// TIA Portal V17 export
// export: Created 2025-05-08T13:17:33.0861985Z, ExportSetting WithDefaults, DisplayName Totally Integrated Automation Portal, DisplayVersion V17 Update 8, DisplayName TIA Portal Openness, DisplayVersion V17 Update 8, DisplayName TIA Portal Version Control Interface, DisplayVersion V17, DisplayName SINAMICS Startdrive Advanced, DisplayVersion V17 SP2, DisplayName SINAMICS Startdrive G110M, G120, G120C, G120D, G120P, G115D, DisplayVersion V17 SP2, DisplayName SINAMICS Startdrive G130, G150, S120, S150, SINAMICS MV, S210, DisplayVersion V17 SP2, DisplayName STEP 7 Professional, DisplayVersion V17 Update 8, DisplayName SINUMERIK ONE STEP 7 Toolbox, DisplayVersion V17 Update 12, DisplayName SINUMERIK 840D sl STEP 7 Toolbox, DisplayVersion V17 Update 12, DisplayName STEP 7 Safety, DisplayVersion V17 Update 6, DisplayName WinCC Advanced, DisplayVersion V17 Update 8
FUNCTION "FC3500_UNIT_2_FIXTURES" : Void   // FC3500, LAD
TITLE = FIXTURE 1
{ S7_Optimized_Access := 'FALSE' }
AUTHOR : ETXETAR
VERSION : 1.0
// stored: AutoNumber false, IsIECCheckEnabled false, SetENOAutomatically false, UDAEnableTagReadback false
   VAR CONSTANT
      FC_NUMBER : DInt := 2500;
   END_VAR
BEGIN

REGION Network 1: CALL FB2500 FIXTURE 1 UNIT 2 CLADDING
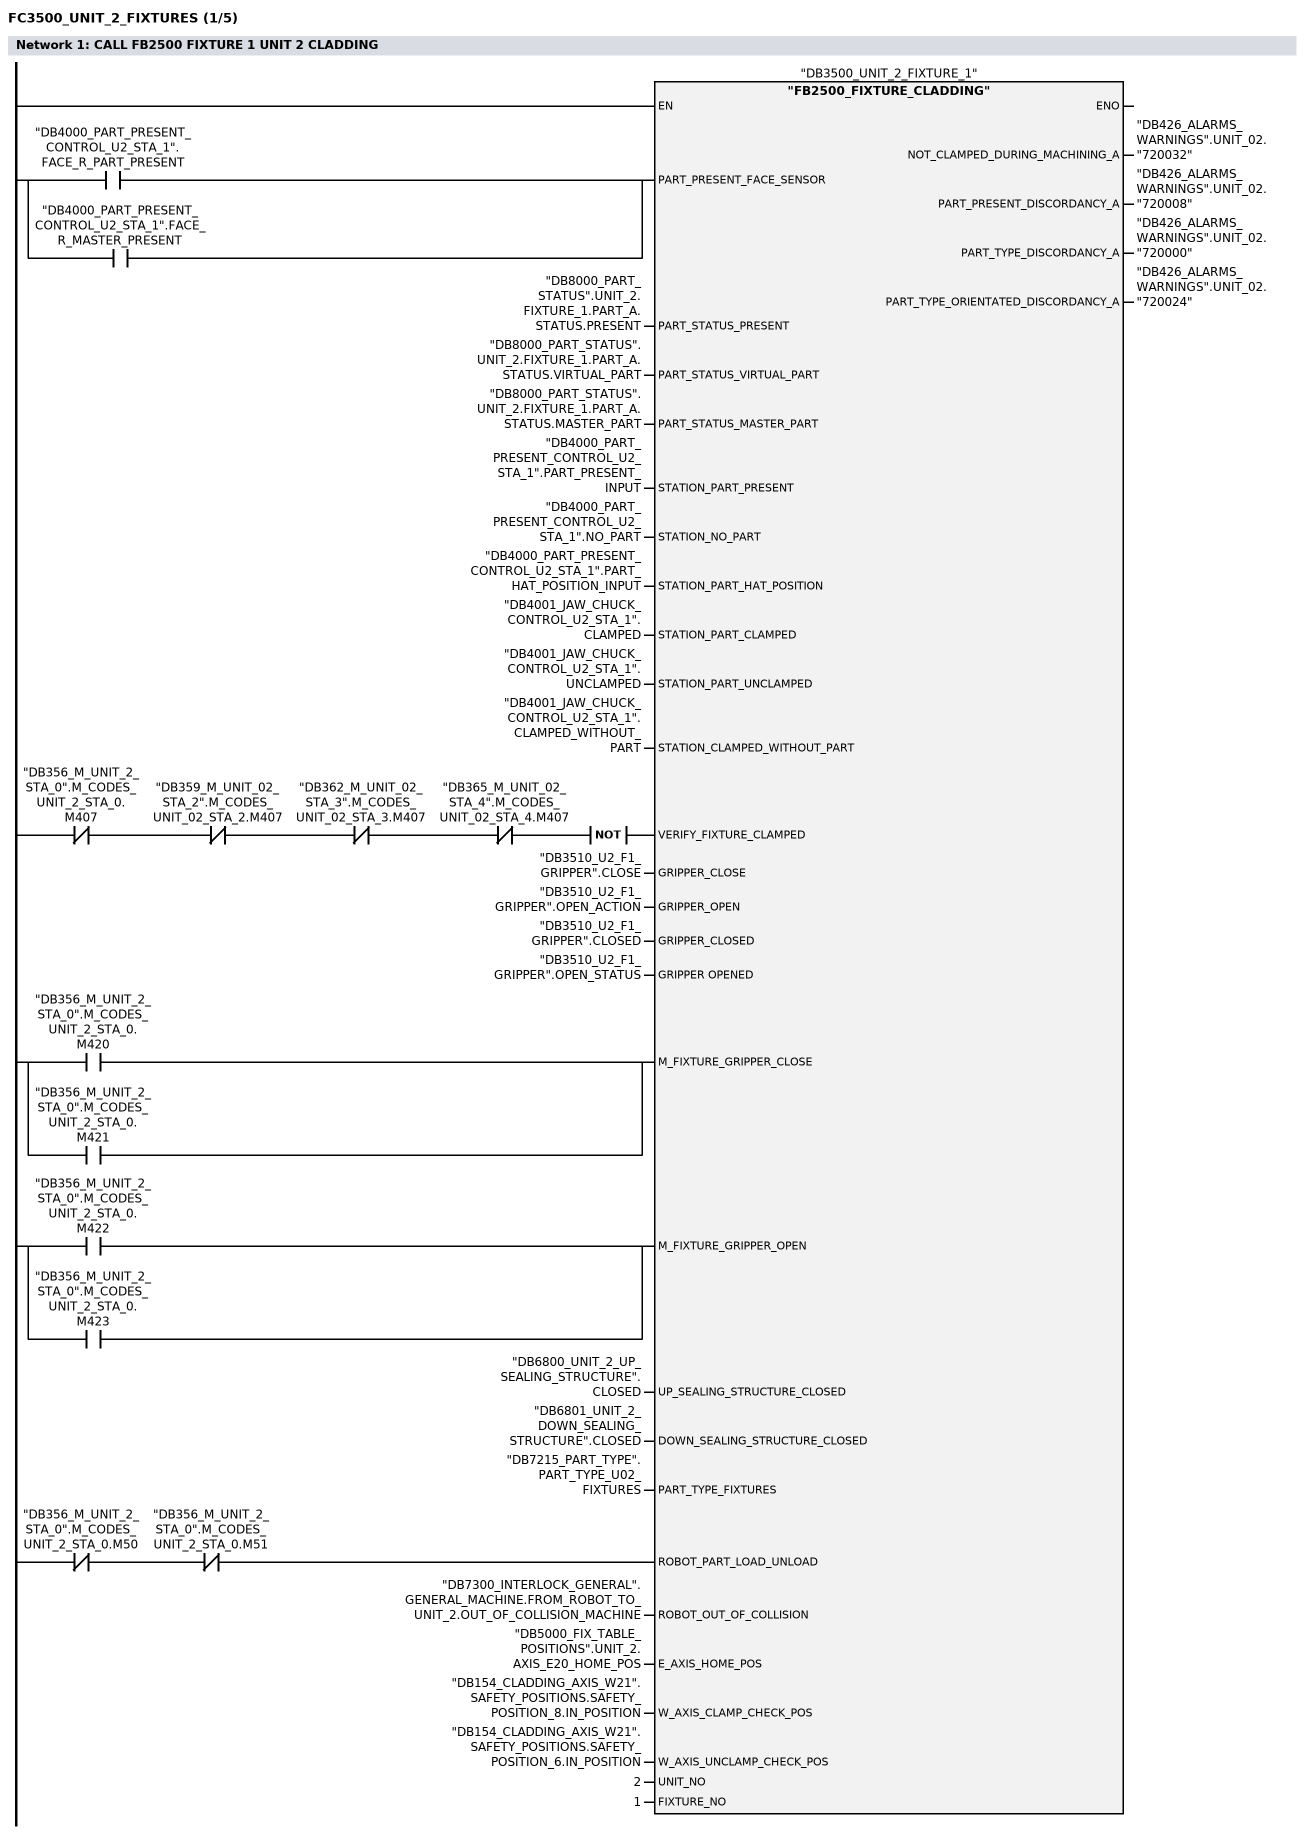
   RUNG wire#powerrail
      "DB3500_UNIT_2_FIXTURE_1"(PART_PRESENT_FACE_SENSOR := wire#w1, VERIFY_FIXTURE_CLAMPED := wire#w2, M_FIXTURE_GRIPPER_CLOSE := wire#w3, M_FIXTURE_GRIPPER_OPEN := wire#w4, ROBOT_PART_LOAD_UNLOAD := wire#w5, PART_STATUS_PRESENT := "DB8000_PART_STATUS".UNIT_2.FIXTURE_1.PART_A.STATUS.PRESENT, PART_STATUS_VIRTUAL_PART := "DB8000_PART_STATUS".UNIT_2.FIXTURE_1.PART_A.STATUS.VIRTUAL_PART, PART_STATUS_MASTER_PART := "DB8000_PART_STATUS".UNIT_2.FIXTURE_1.PART_A.STATUS.MASTER_PART, STATION_PART_PRESENT := "DB4000_PART_PRESENT_CONTROL_U2_STA_1".PART_PRESENT_INPUT, STATION_NO_PART := "DB4000_PART_PRESENT_CONTROL_U2_STA_1".NO_PART, STATION_PART_HAT_POSITION := "DB4000_PART_PRESENT_CONTROL_U2_STA_1".PART_HAT_POSITION_INPUT, STATION_PART_CLAMPED := "DB4001_JAW_CHUCK_CONTROL_U2_STA_1".CLAMPED, STATION_PART_UNCLAMPED := "DB4001_JAW_CHUCK_CONTROL_U2_STA_1".UNCLAMPED, STATION_CLAMPED_WITHOUT_PART := "DB4001_JAW_CHUCK_CONTROL_U2_STA_1".CLAMPED_WITHOUT_PART, GRIPPER_CLOSE := "DB3510_U2_F1_GRIPPER".CLOSE, GRIPPER_OPEN := "DB3510_U2_F1_GRIPPER".OPEN_ACTION, GRIPPER_CLOSED := "DB3510_U2_F1_GRIPPER".CLOSED, "GRIPPER OPENED" := "DB3510_U2_F1_GRIPPER".OPEN_STATUS, UP_SEALING_STRUCTURE_CLOSED := "DB6800_UNIT_2_UP_SEALING_STRUCTURE".CLOSED, DOWN_SEALING_STRUCTURE_CLOSED := "DB6801_UNIT_2_DOWN_SEALING_STRUCTURE".CLOSED, PART_TYPE_FIXTURES := "DB7215_PART_TYPE".PART_TYPE_U02_FIXTURES, ROBOT_OUT_OF_COLLISION := "DB7300_INTERLOCK_GENERAL".GENERAL_MACHINE.FROM_ROBOT_TO_UNIT_2.OUT_OF_COLLISION_MACHINE, E_AXIS_HOME_POS := "DB5000_FIX_TABLE_POSITIONS".UNIT_2.AXIS_E20_HOME_POS, W_AXIS_CLAMP_CHECK_POS := "DB154_CLADDING_AXIS_W21".SAFETY_POSITIONS.SAFETY_POSITION_8.IN_POSITION, W_AXIS_UNCLAMP_CHECK_POS := "DB154_CLADDING_AXIS_W21".SAFETY_POSITIONS.SAFETY_POSITION_6.IN_POSITION, UNIT_NO := 2, FIXTURE_NO := 1, NOT_CLAMPED_DURING_MACHINING_A => "DB426_ALARMS_WARNINGS".UNIT_02."720032", PART_PRESENT_DISCORDANCY_A => "DB426_ALARMS_WARNINGS".UNIT_02."720008", PART_TYPE_DISCORDANCY_A => "DB426_ALARMS_WARNINGS".UNIT_02."720000", PART_TYPE_ORIENTATED_DISCORDANCY_A => "DB426_ALARMS_WARNINGS".UNIT_02."720024")
   END_RUNG
   RUNG wire#powerrail
      Contact( "DB4000_PART_PRESENT_CONTROL_U2_STA_1".FACE_R_PART_PRESENT )
   END_RUNG wire#w1
   RUNG wire#powerrail
      Contact( "DB4000_PART_PRESENT_CONTROL_U2_STA_1".FACE_R_MASTER_PRESENT )
   END_RUNG wire#w1
   RUNG wire#powerrail
      I_Contact( "DB356_M_UNIT_2_STA_0".M_CODES_UNIT_2_STA_0.M407 )
      I_Contact( "DB359_M_UNIT_02_STA_2".M_CODES_UNIT_02_STA_2.M407 )
      I_Contact( "DB362_M_UNIT_02_STA_3".M_CODES_UNIT_02_STA_3.M407 )
      I_Contact( "DB365_M_UNIT_02_STA_4".M_CODES_UNIT_02_STA_4.M407 )
      Not()
   END_RUNG wire#w2
   RUNG wire#powerrail
      Contact( "DB356_M_UNIT_2_STA_0".M_CODES_UNIT_2_STA_0.M420 )
   END_RUNG wire#w3
   RUNG wire#powerrail
      Contact( "DB356_M_UNIT_2_STA_0".M_CODES_UNIT_2_STA_0.M421 )
   END_RUNG wire#w3
   RUNG wire#powerrail
      Contact( "DB356_M_UNIT_2_STA_0".M_CODES_UNIT_2_STA_0.M422 )
   END_RUNG wire#w4
   RUNG wire#powerrail
      Contact( "DB356_M_UNIT_2_STA_0".M_CODES_UNIT_2_STA_0.M423 )
   END_RUNG wire#w4
   RUNG wire#powerrail
      I_Contact( "DB356_M_UNIT_2_STA_0".M_CODES_UNIT_2_STA_0.M50 )
      I_Contact( "DB356_M_UNIT_2_STA_0".M_CODES_UNIT_2_STA_0.M51 )
   END_RUNG wire#w5
   // the same network as SCL:
   "DB3500_UNIT_2_FIXTURE_1"(PART_PRESENT_FACE_SENSOR := "DB4000_PART_PRESENT_CONTROL_U2_STA_1".FACE_R_PART_PRESENT OR "DB4000_PART_PRESENT_CONTROL_U2_STA_1".FACE_R_MASTER_PRESENT,   // "FB2500_FIXTURE_CLADDING"
                           PART_STATUS_PRESENT := "DB8000_PART_STATUS".UNIT_2.FIXTURE_1.PART_A.STATUS.PRESENT,
                           PART_STATUS_VIRTUAL_PART := "DB8000_PART_STATUS".UNIT_2.FIXTURE_1.PART_A.STATUS.VIRTUAL_PART,
                           PART_STATUS_MASTER_PART := "DB8000_PART_STATUS".UNIT_2.FIXTURE_1.PART_A.STATUS.MASTER_PART,
                           STATION_PART_PRESENT := "DB4000_PART_PRESENT_CONTROL_U2_STA_1".PART_PRESENT_INPUT,
                           STATION_NO_PART := "DB4000_PART_PRESENT_CONTROL_U2_STA_1".NO_PART,
                           STATION_PART_HAT_POSITION := "DB4000_PART_PRESENT_CONTROL_U2_STA_1".PART_HAT_POSITION_INPUT,
                           STATION_PART_CLAMPED := "DB4001_JAW_CHUCK_CONTROL_U2_STA_1".CLAMPED,
                           STATION_PART_UNCLAMPED := "DB4001_JAW_CHUCK_CONTROL_U2_STA_1".UNCLAMPED,
                           STATION_CLAMPED_WITHOUT_PART := "DB4001_JAW_CHUCK_CONTROL_U2_STA_1".CLAMPED_WITHOUT_PART,
                           VERIFY_FIXTURE_CLAMPED := NOT (NOT "DB356_M_UNIT_2_STA_0".M_CODES_UNIT_2_STA_0.M407 AND NOT "DB359_M_UNIT_02_STA_2".M_CODES_UNIT_02_STA_2.M407 AND NOT "DB362_M_UNIT_02_STA_3".M_CODES_UNIT_02_STA_3.M407 AND NOT "DB365_M_UNIT_02_STA_4".M_CODES_UNIT_02_STA_4.M407),
                           GRIPPER_CLOSE := "DB3510_U2_F1_GRIPPER".CLOSE,
                           GRIPPER_OPEN := "DB3510_U2_F1_GRIPPER".OPEN_ACTION,
                           GRIPPER_CLOSED := "DB3510_U2_F1_GRIPPER".CLOSED,
                           "GRIPPER OPENED" := "DB3510_U2_F1_GRIPPER".OPEN_STATUS,
                           M_FIXTURE_GRIPPER_CLOSE := "DB356_M_UNIT_2_STA_0".M_CODES_UNIT_2_STA_0.M420 OR "DB356_M_UNIT_2_STA_0".M_CODES_UNIT_2_STA_0.M421,
                           M_FIXTURE_GRIPPER_OPEN := "DB356_M_UNIT_2_STA_0".M_CODES_UNIT_2_STA_0.M422 OR "DB356_M_UNIT_2_STA_0".M_CODES_UNIT_2_STA_0.M423,
                           UP_SEALING_STRUCTURE_CLOSED := "DB6800_UNIT_2_UP_SEALING_STRUCTURE".CLOSED,
                           DOWN_SEALING_STRUCTURE_CLOSED := "DB6801_UNIT_2_DOWN_SEALING_STRUCTURE".CLOSED,
                           PART_TYPE_FIXTURES := "DB7215_PART_TYPE".PART_TYPE_U02_FIXTURES,
                           ROBOT_PART_LOAD_UNLOAD := NOT "DB356_M_UNIT_2_STA_0".M_CODES_UNIT_2_STA_0.M50 AND NOT "DB356_M_UNIT_2_STA_0".M_CODES_UNIT_2_STA_0.M51,
                           ROBOT_OUT_OF_COLLISION := "DB7300_INTERLOCK_GENERAL".GENERAL_MACHINE.FROM_ROBOT_TO_UNIT_2.OUT_OF_COLLISION_MACHINE,
                           E_AXIS_HOME_POS := "DB5000_FIX_TABLE_POSITIONS".UNIT_2.AXIS_E20_HOME_POS,
                           W_AXIS_CLAMP_CHECK_POS := "DB154_CLADDING_AXIS_W21".SAFETY_POSITIONS.SAFETY_POSITION_8.IN_POSITION,
                           W_AXIS_UNCLAMP_CHECK_POS := "DB154_CLADDING_AXIS_W21".SAFETY_POSITIONS.SAFETY_POSITION_6.IN_POSITION,
                           UNIT_NO := 2,
                           FIXTURE_NO := 1,
                           NOT_CLAMPED_DURING_MACHINING_A => "DB426_ALARMS_WARNINGS".UNIT_02."720032",
                           PART_PRESENT_DISCORDANCY_A => "DB426_ALARMS_WARNINGS".UNIT_02."720008",
                           PART_TYPE_DISCORDANCY_A => "DB426_ALARMS_WARNINGS".UNIT_02."720000",
                           PART_TYPE_ORIENTATED_DISCORDANCY_A => "DB426_ALARMS_WARNINGS".UNIT_02."720024");
END_REGION

REGION Network 2: CALL FB2600 FIXTURE 2 UNIT 2 CLADDING
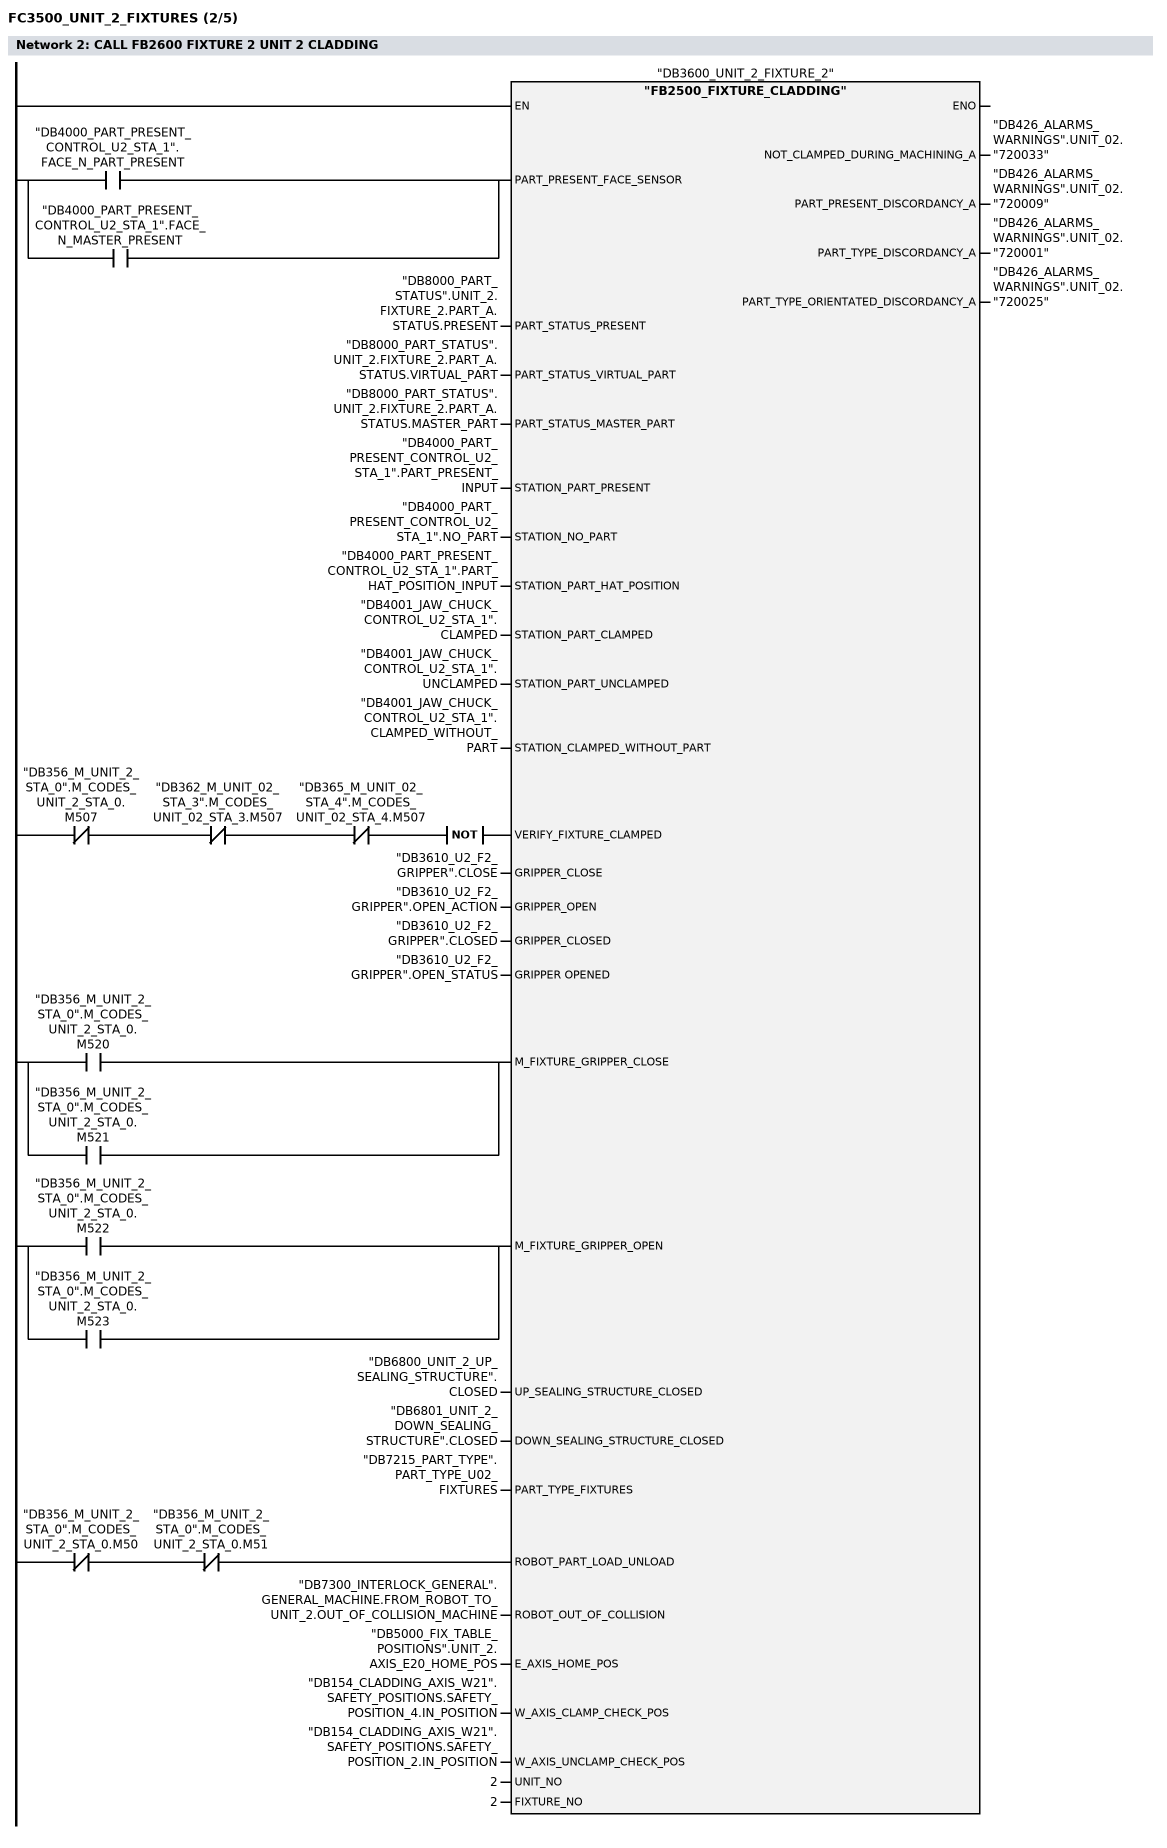
   RUNG wire#powerrail
      "DB3600_UNIT_2_FIXTURE_2"(PART_PRESENT_FACE_SENSOR := wire#w1, VERIFY_FIXTURE_CLAMPED := wire#w2, M_FIXTURE_GRIPPER_CLOSE := wire#w3, M_FIXTURE_GRIPPER_OPEN := wire#w4, ROBOT_PART_LOAD_UNLOAD := wire#w5, PART_STATUS_PRESENT := "DB8000_PART_STATUS".UNIT_2.FIXTURE_2.PART_A.STATUS.PRESENT, PART_STATUS_VIRTUAL_PART := "DB8000_PART_STATUS".UNIT_2.FIXTURE_2.PART_A.STATUS.VIRTUAL_PART, PART_STATUS_MASTER_PART := "DB8000_PART_STATUS".UNIT_2.FIXTURE_2.PART_A.STATUS.MASTER_PART, STATION_PART_PRESENT := "DB4000_PART_PRESENT_CONTROL_U2_STA_1".PART_PRESENT_INPUT, STATION_NO_PART := "DB4000_PART_PRESENT_CONTROL_U2_STA_1".NO_PART, STATION_PART_HAT_POSITION := "DB4000_PART_PRESENT_CONTROL_U2_STA_1".PART_HAT_POSITION_INPUT, STATION_PART_CLAMPED := "DB4001_JAW_CHUCK_CONTROL_U2_STA_1".CLAMPED, STATION_PART_UNCLAMPED := "DB4001_JAW_CHUCK_CONTROL_U2_STA_1".UNCLAMPED, STATION_CLAMPED_WITHOUT_PART := "DB4001_JAW_CHUCK_CONTROL_U2_STA_1".CLAMPED_WITHOUT_PART, GRIPPER_CLOSE := "DB3610_U2_F2_GRIPPER".CLOSE, GRIPPER_OPEN := "DB3610_U2_F2_GRIPPER".OPEN_ACTION, GRIPPER_CLOSED := "DB3610_U2_F2_GRIPPER".CLOSED, "GRIPPER OPENED" := "DB3610_U2_F2_GRIPPER".OPEN_STATUS, UP_SEALING_STRUCTURE_CLOSED := "DB6800_UNIT_2_UP_SEALING_STRUCTURE".CLOSED, DOWN_SEALING_STRUCTURE_CLOSED := "DB6801_UNIT_2_DOWN_SEALING_STRUCTURE".CLOSED, PART_TYPE_FIXTURES := "DB7215_PART_TYPE".PART_TYPE_U02_FIXTURES, ROBOT_OUT_OF_COLLISION := "DB7300_INTERLOCK_GENERAL".GENERAL_MACHINE.FROM_ROBOT_TO_UNIT_2.OUT_OF_COLLISION_MACHINE, E_AXIS_HOME_POS := "DB5000_FIX_TABLE_POSITIONS".UNIT_2.AXIS_E20_HOME_POS, W_AXIS_CLAMP_CHECK_POS := "DB154_CLADDING_AXIS_W21".SAFETY_POSITIONS.SAFETY_POSITION_4.IN_POSITION, W_AXIS_UNCLAMP_CHECK_POS := "DB154_CLADDING_AXIS_W21".SAFETY_POSITIONS.SAFETY_POSITION_2.IN_POSITION, UNIT_NO := 2, FIXTURE_NO := 2, NOT_CLAMPED_DURING_MACHINING_A => "DB426_ALARMS_WARNINGS".UNIT_02."720033", PART_PRESENT_DISCORDANCY_A => "DB426_ALARMS_WARNINGS".UNIT_02."720009", PART_TYPE_DISCORDANCY_A => "DB426_ALARMS_WARNINGS".UNIT_02."720001", PART_TYPE_ORIENTATED_DISCORDANCY_A => "DB426_ALARMS_WARNINGS".UNIT_02."720025")
   END_RUNG
   RUNG wire#powerrail
      Contact( "DB4000_PART_PRESENT_CONTROL_U2_STA_1".FACE_N_PART_PRESENT )
   END_RUNG wire#w1
   RUNG wire#powerrail
      Contact( "DB4000_PART_PRESENT_CONTROL_U2_STA_1".FACE_N_MASTER_PRESENT )
   END_RUNG wire#w1
   RUNG wire#powerrail
      I_Contact( "DB356_M_UNIT_2_STA_0".M_CODES_UNIT_2_STA_0.M507 )
      I_Contact( "DB362_M_UNIT_02_STA_3".M_CODES_UNIT_02_STA_3.M507 )
      I_Contact( "DB365_M_UNIT_02_STA_4".M_CODES_UNIT_02_STA_4.M507 )
      Not()
   END_RUNG wire#w2
   RUNG wire#powerrail
      Contact( "DB356_M_UNIT_2_STA_0".M_CODES_UNIT_2_STA_0.M520 )
   END_RUNG wire#w3
   RUNG wire#powerrail
      Contact( "DB356_M_UNIT_2_STA_0".M_CODES_UNIT_2_STA_0.M521 )
   END_RUNG wire#w3
   RUNG wire#powerrail
      Contact( "DB356_M_UNIT_2_STA_0".M_CODES_UNIT_2_STA_0.M522 )
   END_RUNG wire#w4
   RUNG wire#powerrail
      Contact( "DB356_M_UNIT_2_STA_0".M_CODES_UNIT_2_STA_0.M523 )
   END_RUNG wire#w4
   RUNG wire#powerrail
      I_Contact( "DB356_M_UNIT_2_STA_0".M_CODES_UNIT_2_STA_0.M50 )
      I_Contact( "DB356_M_UNIT_2_STA_0".M_CODES_UNIT_2_STA_0.M51 )
   END_RUNG wire#w5
   // the same network as SCL:
   "DB3600_UNIT_2_FIXTURE_2"(PART_PRESENT_FACE_SENSOR := "DB4000_PART_PRESENT_CONTROL_U2_STA_1".FACE_N_PART_PRESENT OR "DB4000_PART_PRESENT_CONTROL_U2_STA_1".FACE_N_MASTER_PRESENT,   // "FB2500_FIXTURE_CLADDING"
                           PART_STATUS_PRESENT := "DB8000_PART_STATUS".UNIT_2.FIXTURE_2.PART_A.STATUS.PRESENT,
                           PART_STATUS_VIRTUAL_PART := "DB8000_PART_STATUS".UNIT_2.FIXTURE_2.PART_A.STATUS.VIRTUAL_PART,
                           PART_STATUS_MASTER_PART := "DB8000_PART_STATUS".UNIT_2.FIXTURE_2.PART_A.STATUS.MASTER_PART,
                           STATION_PART_PRESENT := "DB4000_PART_PRESENT_CONTROL_U2_STA_1".PART_PRESENT_INPUT,
                           STATION_NO_PART := "DB4000_PART_PRESENT_CONTROL_U2_STA_1".NO_PART,
                           STATION_PART_HAT_POSITION := "DB4000_PART_PRESENT_CONTROL_U2_STA_1".PART_HAT_POSITION_INPUT,
                           STATION_PART_CLAMPED := "DB4001_JAW_CHUCK_CONTROL_U2_STA_1".CLAMPED,
                           STATION_PART_UNCLAMPED := "DB4001_JAW_CHUCK_CONTROL_U2_STA_1".UNCLAMPED,
                           STATION_CLAMPED_WITHOUT_PART := "DB4001_JAW_CHUCK_CONTROL_U2_STA_1".CLAMPED_WITHOUT_PART,
                           VERIFY_FIXTURE_CLAMPED := NOT (NOT "DB356_M_UNIT_2_STA_0".M_CODES_UNIT_2_STA_0.M507 AND NOT "DB362_M_UNIT_02_STA_3".M_CODES_UNIT_02_STA_3.M507 AND NOT "DB365_M_UNIT_02_STA_4".M_CODES_UNIT_02_STA_4.M507),
                           GRIPPER_CLOSE := "DB3610_U2_F2_GRIPPER".CLOSE,
                           GRIPPER_OPEN := "DB3610_U2_F2_GRIPPER".OPEN_ACTION,
                           GRIPPER_CLOSED := "DB3610_U2_F2_GRIPPER".CLOSED,
                           "GRIPPER OPENED" := "DB3610_U2_F2_GRIPPER".OPEN_STATUS,
                           M_FIXTURE_GRIPPER_CLOSE := "DB356_M_UNIT_2_STA_0".M_CODES_UNIT_2_STA_0.M520 OR "DB356_M_UNIT_2_STA_0".M_CODES_UNIT_2_STA_0.M521,
                           M_FIXTURE_GRIPPER_OPEN := "DB356_M_UNIT_2_STA_0".M_CODES_UNIT_2_STA_0.M522 OR "DB356_M_UNIT_2_STA_0".M_CODES_UNIT_2_STA_0.M523,
                           UP_SEALING_STRUCTURE_CLOSED := "DB6800_UNIT_2_UP_SEALING_STRUCTURE".CLOSED,
                           DOWN_SEALING_STRUCTURE_CLOSED := "DB6801_UNIT_2_DOWN_SEALING_STRUCTURE".CLOSED,
                           PART_TYPE_FIXTURES := "DB7215_PART_TYPE".PART_TYPE_U02_FIXTURES,
                           ROBOT_PART_LOAD_UNLOAD := NOT "DB356_M_UNIT_2_STA_0".M_CODES_UNIT_2_STA_0.M50 AND NOT "DB356_M_UNIT_2_STA_0".M_CODES_UNIT_2_STA_0.M51,
                           ROBOT_OUT_OF_COLLISION := "DB7300_INTERLOCK_GENERAL".GENERAL_MACHINE.FROM_ROBOT_TO_UNIT_2.OUT_OF_COLLISION_MACHINE,
                           E_AXIS_HOME_POS := "DB5000_FIX_TABLE_POSITIONS".UNIT_2.AXIS_E20_HOME_POS,
                           W_AXIS_CLAMP_CHECK_POS := "DB154_CLADDING_AXIS_W21".SAFETY_POSITIONS.SAFETY_POSITION_4.IN_POSITION,
                           W_AXIS_UNCLAMP_CHECK_POS := "DB154_CLADDING_AXIS_W21".SAFETY_POSITIONS.SAFETY_POSITION_2.IN_POSITION,
                           UNIT_NO := 2,
                           FIXTURE_NO := 2,
                           NOT_CLAMPED_DURING_MACHINING_A => "DB426_ALARMS_WARNINGS".UNIT_02."720033",
                           PART_PRESENT_DISCORDANCY_A => "DB426_ALARMS_WARNINGS".UNIT_02."720009",
                           PART_TYPE_DISCORDANCY_A => "DB426_ALARMS_WARNINGS".UNIT_02."720001",
                           PART_TYPE_ORIENTATED_DISCORDANCY_A => "DB426_ALARMS_WARNINGS".UNIT_02."720025");
END_REGION

REGION Network 3: CALL FB2600 FIXTURE 3 UNIT 2 CLADDING
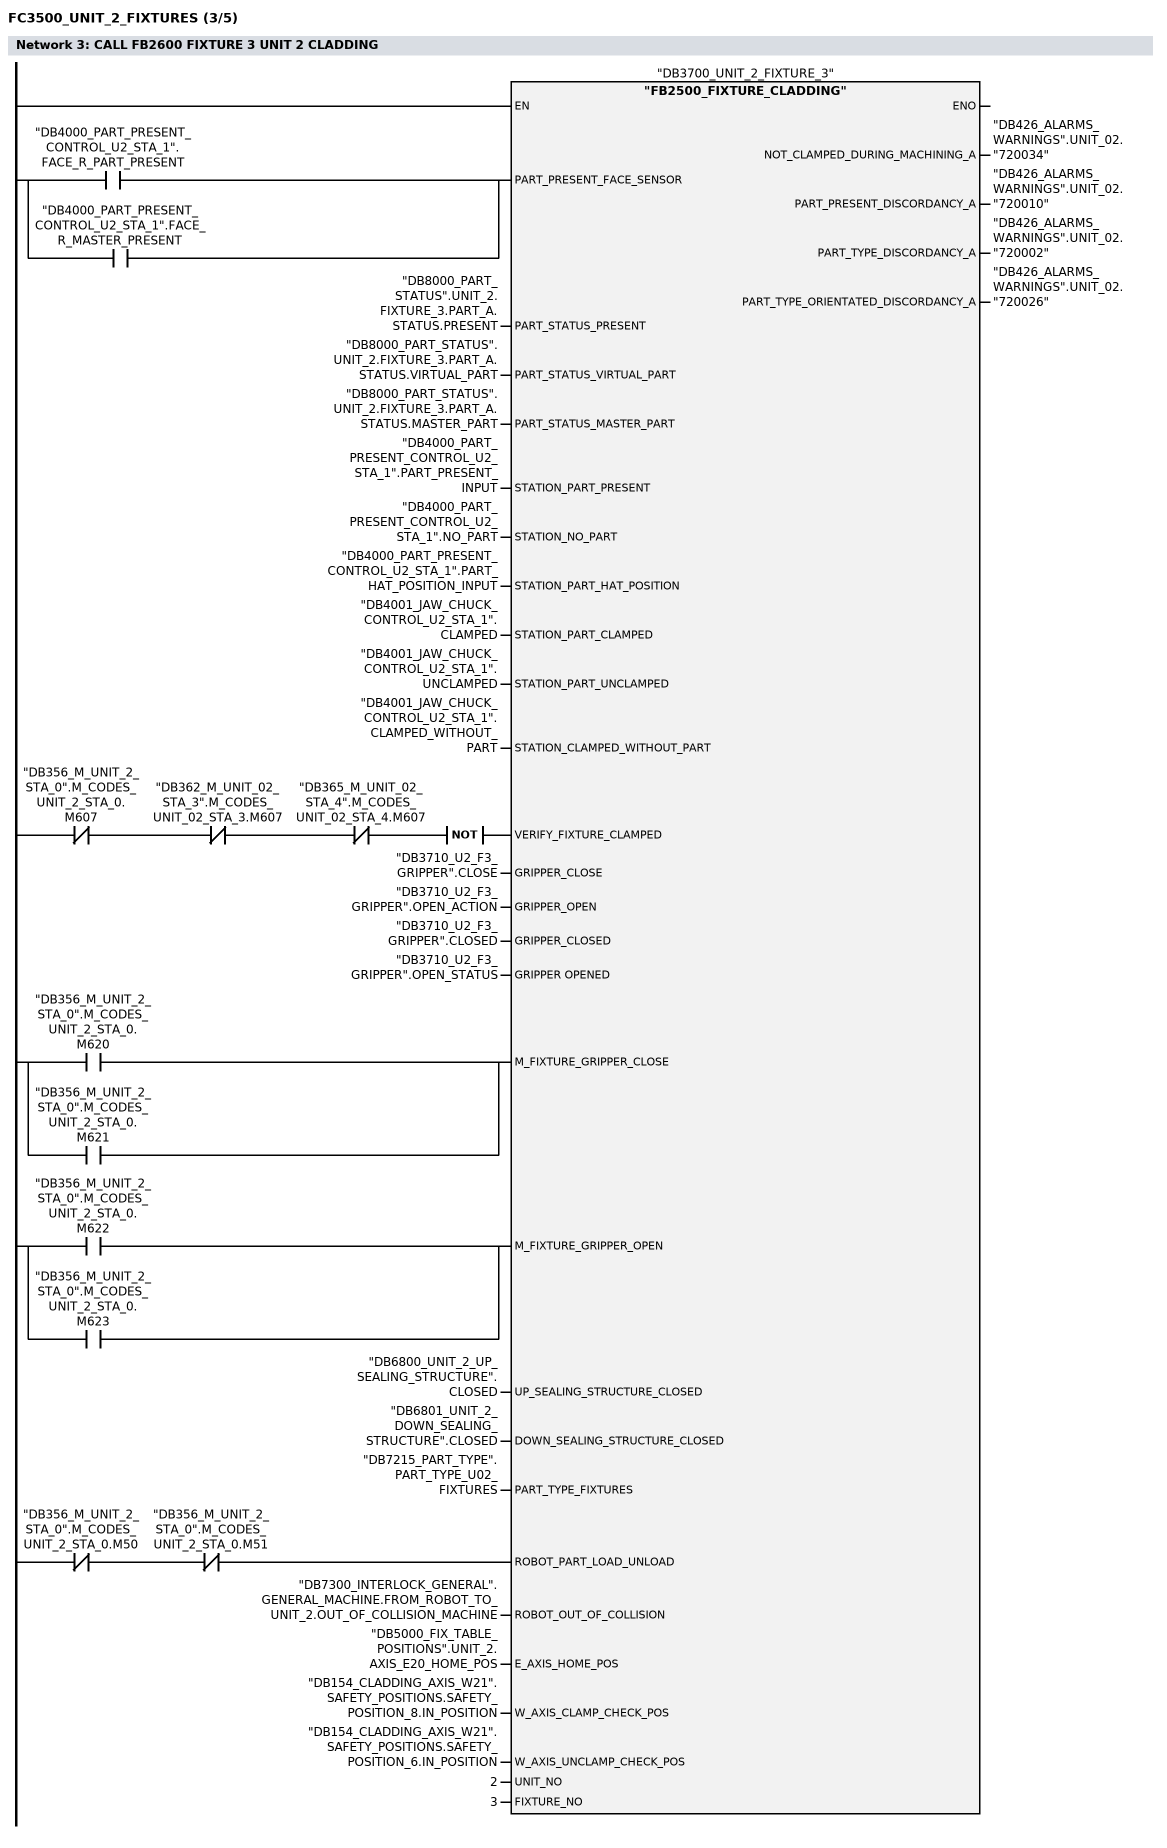
   RUNG wire#powerrail
      "DB3700_UNIT_2_FIXTURE_3"(PART_PRESENT_FACE_SENSOR := wire#w1, VERIFY_FIXTURE_CLAMPED := wire#w2, M_FIXTURE_GRIPPER_CLOSE := wire#w3, M_FIXTURE_GRIPPER_OPEN := wire#w4, ROBOT_PART_LOAD_UNLOAD := wire#w5, PART_STATUS_PRESENT := "DB8000_PART_STATUS".UNIT_2.FIXTURE_3.PART_A.STATUS.PRESENT, PART_STATUS_VIRTUAL_PART := "DB8000_PART_STATUS".UNIT_2.FIXTURE_3.PART_A.STATUS.VIRTUAL_PART, PART_STATUS_MASTER_PART := "DB8000_PART_STATUS".UNIT_2.FIXTURE_3.PART_A.STATUS.MASTER_PART, STATION_PART_PRESENT := "DB4000_PART_PRESENT_CONTROL_U2_STA_1".PART_PRESENT_INPUT, STATION_NO_PART := "DB4000_PART_PRESENT_CONTROL_U2_STA_1".NO_PART, STATION_PART_HAT_POSITION := "DB4000_PART_PRESENT_CONTROL_U2_STA_1".PART_HAT_POSITION_INPUT, STATION_PART_CLAMPED := "DB4001_JAW_CHUCK_CONTROL_U2_STA_1".CLAMPED, STATION_PART_UNCLAMPED := "DB4001_JAW_CHUCK_CONTROL_U2_STA_1".UNCLAMPED, STATION_CLAMPED_WITHOUT_PART := "DB4001_JAW_CHUCK_CONTROL_U2_STA_1".CLAMPED_WITHOUT_PART, GRIPPER_CLOSE := "DB3710_U2_F3_GRIPPER".CLOSE, GRIPPER_OPEN := "DB3710_U2_F3_GRIPPER".OPEN_ACTION, GRIPPER_CLOSED := "DB3710_U2_F3_GRIPPER".CLOSED, "GRIPPER OPENED" := "DB3710_U2_F3_GRIPPER".OPEN_STATUS, UP_SEALING_STRUCTURE_CLOSED := "DB6800_UNIT_2_UP_SEALING_STRUCTURE".CLOSED, DOWN_SEALING_STRUCTURE_CLOSED := "DB6801_UNIT_2_DOWN_SEALING_STRUCTURE".CLOSED, PART_TYPE_FIXTURES := "DB7215_PART_TYPE".PART_TYPE_U02_FIXTURES, ROBOT_OUT_OF_COLLISION := "DB7300_INTERLOCK_GENERAL".GENERAL_MACHINE.FROM_ROBOT_TO_UNIT_2.OUT_OF_COLLISION_MACHINE, E_AXIS_HOME_POS := "DB5000_FIX_TABLE_POSITIONS".UNIT_2.AXIS_E20_HOME_POS, W_AXIS_CLAMP_CHECK_POS := "DB154_CLADDING_AXIS_W21".SAFETY_POSITIONS.SAFETY_POSITION_8.IN_POSITION, W_AXIS_UNCLAMP_CHECK_POS := "DB154_CLADDING_AXIS_W21".SAFETY_POSITIONS.SAFETY_POSITION_6.IN_POSITION, UNIT_NO := 2, FIXTURE_NO := 3, NOT_CLAMPED_DURING_MACHINING_A => "DB426_ALARMS_WARNINGS".UNIT_02."720034", PART_PRESENT_DISCORDANCY_A => "DB426_ALARMS_WARNINGS".UNIT_02."720010", PART_TYPE_DISCORDANCY_A => "DB426_ALARMS_WARNINGS".UNIT_02."720002", PART_TYPE_ORIENTATED_DISCORDANCY_A => "DB426_ALARMS_WARNINGS".UNIT_02."720026")
   END_RUNG
   RUNG wire#powerrail
      Contact( "DB4000_PART_PRESENT_CONTROL_U2_STA_1".FACE_R_PART_PRESENT )
   END_RUNG wire#w1
   RUNG wire#powerrail
      Contact( "DB4000_PART_PRESENT_CONTROL_U2_STA_1".FACE_R_MASTER_PRESENT )
   END_RUNG wire#w1
   RUNG wire#powerrail
      I_Contact( "DB356_M_UNIT_2_STA_0".M_CODES_UNIT_2_STA_0.M607 )
      I_Contact( "DB362_M_UNIT_02_STA_3".M_CODES_UNIT_02_STA_3.M607 )
      I_Contact( "DB365_M_UNIT_02_STA_4".M_CODES_UNIT_02_STA_4.M607 )
      Not()
   END_RUNG wire#w2
   RUNG wire#powerrail
      Contact( "DB356_M_UNIT_2_STA_0".M_CODES_UNIT_2_STA_0.M620 )
   END_RUNG wire#w3
   RUNG wire#powerrail
      Contact( "DB356_M_UNIT_2_STA_0".M_CODES_UNIT_2_STA_0.M621 )
   END_RUNG wire#w3
   RUNG wire#powerrail
      Contact( "DB356_M_UNIT_2_STA_0".M_CODES_UNIT_2_STA_0.M622 )
   END_RUNG wire#w4
   RUNG wire#powerrail
      Contact( "DB356_M_UNIT_2_STA_0".M_CODES_UNIT_2_STA_0.M623 )
   END_RUNG wire#w4
   RUNG wire#powerrail
      I_Contact( "DB356_M_UNIT_2_STA_0".M_CODES_UNIT_2_STA_0.M50 )
      I_Contact( "DB356_M_UNIT_2_STA_0".M_CODES_UNIT_2_STA_0.M51 )
   END_RUNG wire#w5
   // the same network as SCL:
   "DB3700_UNIT_2_FIXTURE_3"(PART_PRESENT_FACE_SENSOR := "DB4000_PART_PRESENT_CONTROL_U2_STA_1".FACE_R_PART_PRESENT OR "DB4000_PART_PRESENT_CONTROL_U2_STA_1".FACE_R_MASTER_PRESENT,   // "FB2500_FIXTURE_CLADDING"
                           PART_STATUS_PRESENT := "DB8000_PART_STATUS".UNIT_2.FIXTURE_3.PART_A.STATUS.PRESENT,
                           PART_STATUS_VIRTUAL_PART := "DB8000_PART_STATUS".UNIT_2.FIXTURE_3.PART_A.STATUS.VIRTUAL_PART,
                           PART_STATUS_MASTER_PART := "DB8000_PART_STATUS".UNIT_2.FIXTURE_3.PART_A.STATUS.MASTER_PART,
                           STATION_PART_PRESENT := "DB4000_PART_PRESENT_CONTROL_U2_STA_1".PART_PRESENT_INPUT,
                           STATION_NO_PART := "DB4000_PART_PRESENT_CONTROL_U2_STA_1".NO_PART,
                           STATION_PART_HAT_POSITION := "DB4000_PART_PRESENT_CONTROL_U2_STA_1".PART_HAT_POSITION_INPUT,
                           STATION_PART_CLAMPED := "DB4001_JAW_CHUCK_CONTROL_U2_STA_1".CLAMPED,
                           STATION_PART_UNCLAMPED := "DB4001_JAW_CHUCK_CONTROL_U2_STA_1".UNCLAMPED,
                           STATION_CLAMPED_WITHOUT_PART := "DB4001_JAW_CHUCK_CONTROL_U2_STA_1".CLAMPED_WITHOUT_PART,
                           VERIFY_FIXTURE_CLAMPED := NOT (NOT "DB356_M_UNIT_2_STA_0".M_CODES_UNIT_2_STA_0.M607 AND NOT "DB362_M_UNIT_02_STA_3".M_CODES_UNIT_02_STA_3.M607 AND NOT "DB365_M_UNIT_02_STA_4".M_CODES_UNIT_02_STA_4.M607),
                           GRIPPER_CLOSE := "DB3710_U2_F3_GRIPPER".CLOSE,
                           GRIPPER_OPEN := "DB3710_U2_F3_GRIPPER".OPEN_ACTION,
                           GRIPPER_CLOSED := "DB3710_U2_F3_GRIPPER".CLOSED,
                           "GRIPPER OPENED" := "DB3710_U2_F3_GRIPPER".OPEN_STATUS,
                           M_FIXTURE_GRIPPER_CLOSE := "DB356_M_UNIT_2_STA_0".M_CODES_UNIT_2_STA_0.M620 OR "DB356_M_UNIT_2_STA_0".M_CODES_UNIT_2_STA_0.M621,
                           M_FIXTURE_GRIPPER_OPEN := "DB356_M_UNIT_2_STA_0".M_CODES_UNIT_2_STA_0.M622 OR "DB356_M_UNIT_2_STA_0".M_CODES_UNIT_2_STA_0.M623,
                           UP_SEALING_STRUCTURE_CLOSED := "DB6800_UNIT_2_UP_SEALING_STRUCTURE".CLOSED,
                           DOWN_SEALING_STRUCTURE_CLOSED := "DB6801_UNIT_2_DOWN_SEALING_STRUCTURE".CLOSED,
                           PART_TYPE_FIXTURES := "DB7215_PART_TYPE".PART_TYPE_U02_FIXTURES,
                           ROBOT_PART_LOAD_UNLOAD := NOT "DB356_M_UNIT_2_STA_0".M_CODES_UNIT_2_STA_0.M50 AND NOT "DB356_M_UNIT_2_STA_0".M_CODES_UNIT_2_STA_0.M51,
                           ROBOT_OUT_OF_COLLISION := "DB7300_INTERLOCK_GENERAL".GENERAL_MACHINE.FROM_ROBOT_TO_UNIT_2.OUT_OF_COLLISION_MACHINE,
                           E_AXIS_HOME_POS := "DB5000_FIX_TABLE_POSITIONS".UNIT_2.AXIS_E20_HOME_POS,
                           W_AXIS_CLAMP_CHECK_POS := "DB154_CLADDING_AXIS_W21".SAFETY_POSITIONS.SAFETY_POSITION_8.IN_POSITION,
                           W_AXIS_UNCLAMP_CHECK_POS := "DB154_CLADDING_AXIS_W21".SAFETY_POSITIONS.SAFETY_POSITION_6.IN_POSITION,
                           UNIT_NO := 2,
                           FIXTURE_NO := 3,
                           NOT_CLAMPED_DURING_MACHINING_A => "DB426_ALARMS_WARNINGS".UNIT_02."720034",
                           PART_PRESENT_DISCORDANCY_A => "DB426_ALARMS_WARNINGS".UNIT_02."720010",
                           PART_TYPE_DISCORDANCY_A => "DB426_ALARMS_WARNINGS".UNIT_02."720002",
                           PART_TYPE_ORIENTATED_DISCORDANCY_A => "DB426_ALARMS_WARNINGS".UNIT_02."720026");
END_REGION

REGION Network 4: CALL FB2600 FIXTURE 4 UNIT 2 CLADDING
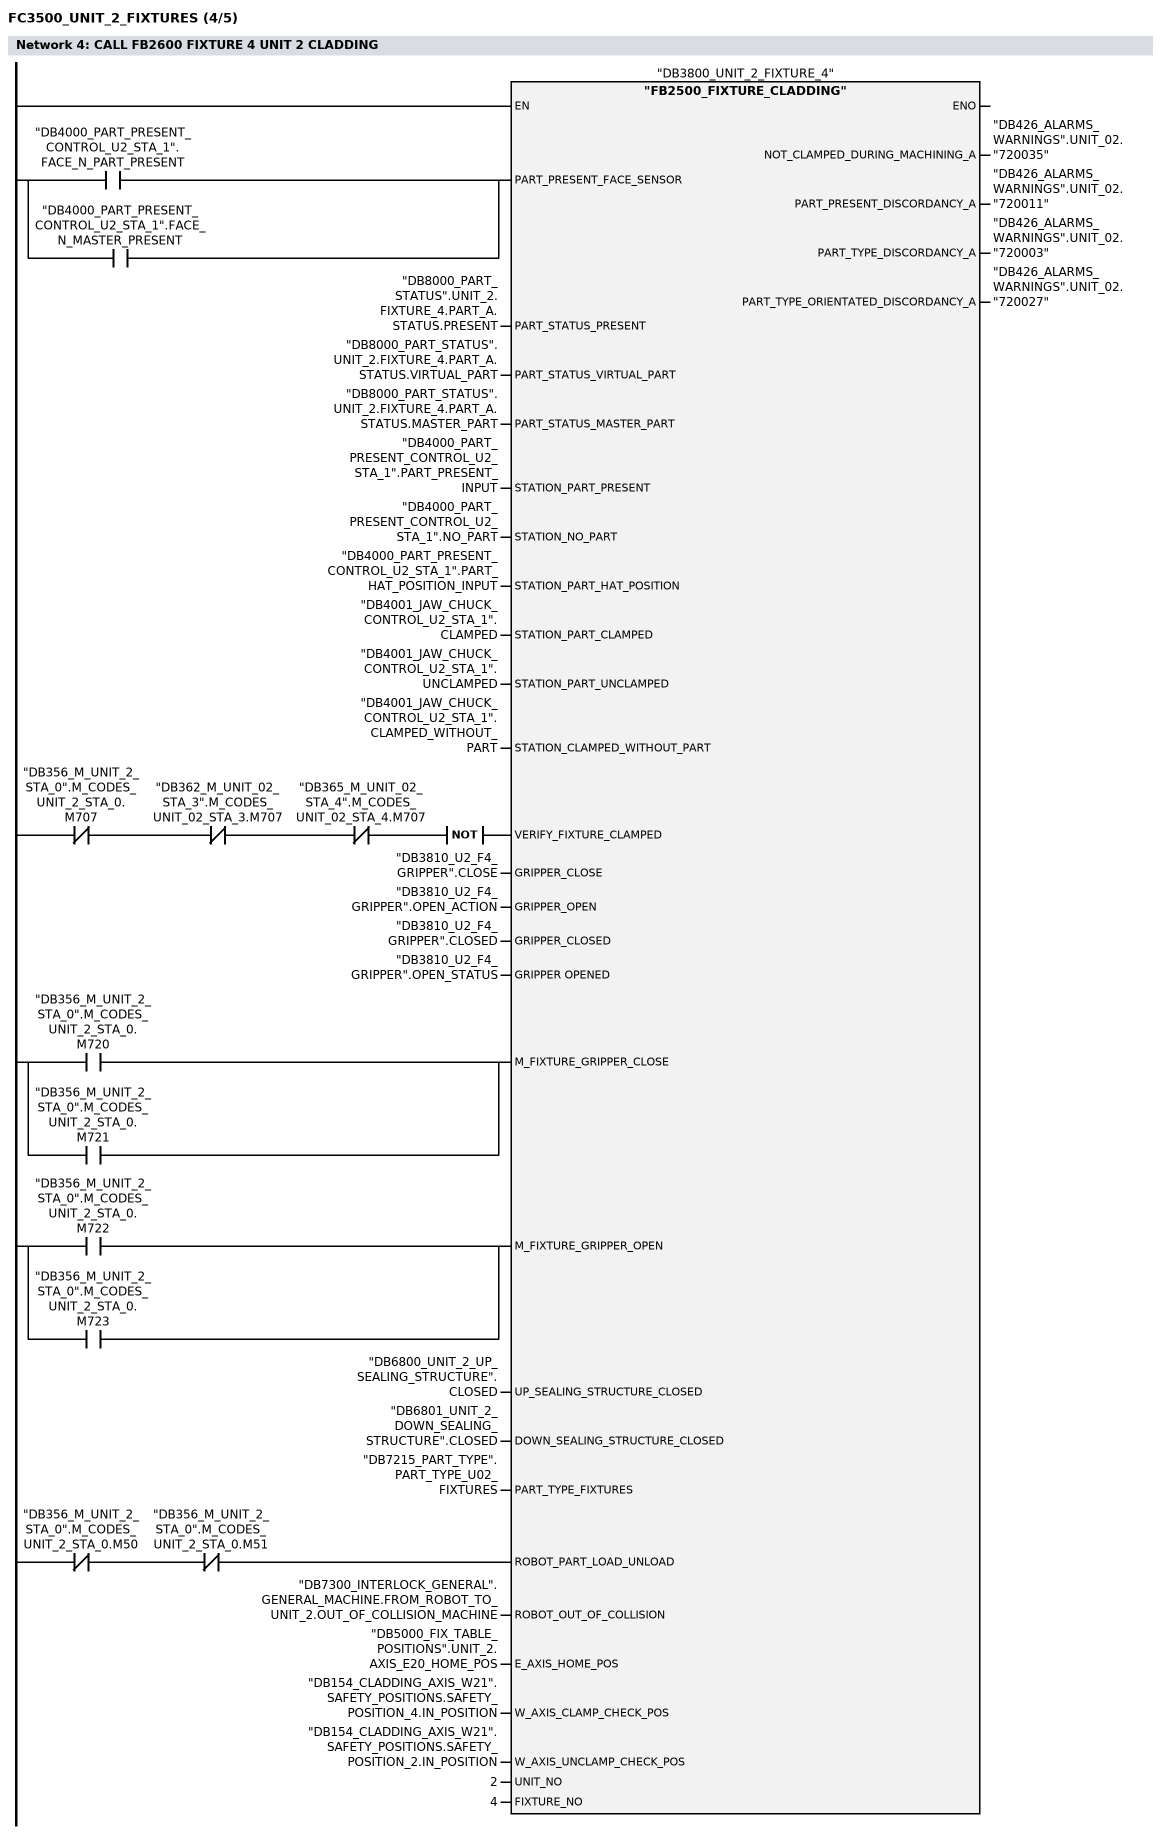
   RUNG wire#powerrail
      "DB3800_UNIT_2_FIXTURE_4"(PART_PRESENT_FACE_SENSOR := wire#w1, VERIFY_FIXTURE_CLAMPED := wire#w2, M_FIXTURE_GRIPPER_CLOSE := wire#w3, M_FIXTURE_GRIPPER_OPEN := wire#w4, ROBOT_PART_LOAD_UNLOAD := wire#w5, PART_STATUS_PRESENT := "DB8000_PART_STATUS".UNIT_2.FIXTURE_4.PART_A.STATUS.PRESENT, PART_STATUS_VIRTUAL_PART := "DB8000_PART_STATUS".UNIT_2.FIXTURE_4.PART_A.STATUS.VIRTUAL_PART, PART_STATUS_MASTER_PART := "DB8000_PART_STATUS".UNIT_2.FIXTURE_4.PART_A.STATUS.MASTER_PART, STATION_PART_PRESENT := "DB4000_PART_PRESENT_CONTROL_U2_STA_1".PART_PRESENT_INPUT, STATION_NO_PART := "DB4000_PART_PRESENT_CONTROL_U2_STA_1".NO_PART, STATION_PART_HAT_POSITION := "DB4000_PART_PRESENT_CONTROL_U2_STA_1".PART_HAT_POSITION_INPUT, STATION_PART_CLAMPED := "DB4001_JAW_CHUCK_CONTROL_U2_STA_1".CLAMPED, STATION_PART_UNCLAMPED := "DB4001_JAW_CHUCK_CONTROL_U2_STA_1".UNCLAMPED, STATION_CLAMPED_WITHOUT_PART := "DB4001_JAW_CHUCK_CONTROL_U2_STA_1".CLAMPED_WITHOUT_PART, GRIPPER_CLOSE := "DB3810_U2_F4_GRIPPER".CLOSE, GRIPPER_OPEN := "DB3810_U2_F4_GRIPPER".OPEN_ACTION, GRIPPER_CLOSED := "DB3810_U2_F4_GRIPPER".CLOSED, "GRIPPER OPENED" := "DB3810_U2_F4_GRIPPER".OPEN_STATUS, UP_SEALING_STRUCTURE_CLOSED := "DB6800_UNIT_2_UP_SEALING_STRUCTURE".CLOSED, DOWN_SEALING_STRUCTURE_CLOSED := "DB6801_UNIT_2_DOWN_SEALING_STRUCTURE".CLOSED, PART_TYPE_FIXTURES := "DB7215_PART_TYPE".PART_TYPE_U02_FIXTURES, ROBOT_OUT_OF_COLLISION := "DB7300_INTERLOCK_GENERAL".GENERAL_MACHINE.FROM_ROBOT_TO_UNIT_2.OUT_OF_COLLISION_MACHINE, E_AXIS_HOME_POS := "DB5000_FIX_TABLE_POSITIONS".UNIT_2.AXIS_E20_HOME_POS, W_AXIS_CLAMP_CHECK_POS := "DB154_CLADDING_AXIS_W21".SAFETY_POSITIONS.SAFETY_POSITION_4.IN_POSITION, W_AXIS_UNCLAMP_CHECK_POS := "DB154_CLADDING_AXIS_W21".SAFETY_POSITIONS.SAFETY_POSITION_2.IN_POSITION, UNIT_NO := 2, FIXTURE_NO := 4, NOT_CLAMPED_DURING_MACHINING_A => "DB426_ALARMS_WARNINGS".UNIT_02."720035", PART_PRESENT_DISCORDANCY_A => "DB426_ALARMS_WARNINGS".UNIT_02."720011", PART_TYPE_DISCORDANCY_A => "DB426_ALARMS_WARNINGS".UNIT_02."720003", PART_TYPE_ORIENTATED_DISCORDANCY_A => "DB426_ALARMS_WARNINGS".UNIT_02."720027")
   END_RUNG
   RUNG wire#powerrail
      Contact( "DB4000_PART_PRESENT_CONTROL_U2_STA_1".FACE_N_PART_PRESENT )
   END_RUNG wire#w1
   RUNG wire#powerrail
      Contact( "DB4000_PART_PRESENT_CONTROL_U2_STA_1".FACE_N_MASTER_PRESENT )
   END_RUNG wire#w1
   RUNG wire#powerrail
      I_Contact( "DB356_M_UNIT_2_STA_0".M_CODES_UNIT_2_STA_0.M707 )
      I_Contact( "DB362_M_UNIT_02_STA_3".M_CODES_UNIT_02_STA_3.M707 )
      I_Contact( "DB365_M_UNIT_02_STA_4".M_CODES_UNIT_02_STA_4.M707 )
      Not()
   END_RUNG wire#w2
   RUNG wire#powerrail
      Contact( "DB356_M_UNIT_2_STA_0".M_CODES_UNIT_2_STA_0.M720 )
   END_RUNG wire#w3
   RUNG wire#powerrail
      Contact( "DB356_M_UNIT_2_STA_0".M_CODES_UNIT_2_STA_0.M721 )
   END_RUNG wire#w3
   RUNG wire#powerrail
      Contact( "DB356_M_UNIT_2_STA_0".M_CODES_UNIT_2_STA_0.M722 )
   END_RUNG wire#w4
   RUNG wire#powerrail
      Contact( "DB356_M_UNIT_2_STA_0".M_CODES_UNIT_2_STA_0.M723 )
   END_RUNG wire#w4
   RUNG wire#powerrail
      I_Contact( "DB356_M_UNIT_2_STA_0".M_CODES_UNIT_2_STA_0.M50 )
      I_Contact( "DB356_M_UNIT_2_STA_0".M_CODES_UNIT_2_STA_0.M51 )
   END_RUNG wire#w5
   // the same network as SCL:
   "DB3800_UNIT_2_FIXTURE_4"(PART_PRESENT_FACE_SENSOR := "DB4000_PART_PRESENT_CONTROL_U2_STA_1".FACE_N_PART_PRESENT OR "DB4000_PART_PRESENT_CONTROL_U2_STA_1".FACE_N_MASTER_PRESENT,   // "FB2500_FIXTURE_CLADDING"
                           PART_STATUS_PRESENT := "DB8000_PART_STATUS".UNIT_2.FIXTURE_4.PART_A.STATUS.PRESENT,
                           PART_STATUS_VIRTUAL_PART := "DB8000_PART_STATUS".UNIT_2.FIXTURE_4.PART_A.STATUS.VIRTUAL_PART,
                           PART_STATUS_MASTER_PART := "DB8000_PART_STATUS".UNIT_2.FIXTURE_4.PART_A.STATUS.MASTER_PART,
                           STATION_PART_PRESENT := "DB4000_PART_PRESENT_CONTROL_U2_STA_1".PART_PRESENT_INPUT,
                           STATION_NO_PART := "DB4000_PART_PRESENT_CONTROL_U2_STA_1".NO_PART,
                           STATION_PART_HAT_POSITION := "DB4000_PART_PRESENT_CONTROL_U2_STA_1".PART_HAT_POSITION_INPUT,
                           STATION_PART_CLAMPED := "DB4001_JAW_CHUCK_CONTROL_U2_STA_1".CLAMPED,
                           STATION_PART_UNCLAMPED := "DB4001_JAW_CHUCK_CONTROL_U2_STA_1".UNCLAMPED,
                           STATION_CLAMPED_WITHOUT_PART := "DB4001_JAW_CHUCK_CONTROL_U2_STA_1".CLAMPED_WITHOUT_PART,
                           VERIFY_FIXTURE_CLAMPED := NOT (NOT "DB356_M_UNIT_2_STA_0".M_CODES_UNIT_2_STA_0.M707 AND NOT "DB362_M_UNIT_02_STA_3".M_CODES_UNIT_02_STA_3.M707 AND NOT "DB365_M_UNIT_02_STA_4".M_CODES_UNIT_02_STA_4.M707),
                           GRIPPER_CLOSE := "DB3810_U2_F4_GRIPPER".CLOSE,
                           GRIPPER_OPEN := "DB3810_U2_F4_GRIPPER".OPEN_ACTION,
                           GRIPPER_CLOSED := "DB3810_U2_F4_GRIPPER".CLOSED,
                           "GRIPPER OPENED" := "DB3810_U2_F4_GRIPPER".OPEN_STATUS,
                           M_FIXTURE_GRIPPER_CLOSE := "DB356_M_UNIT_2_STA_0".M_CODES_UNIT_2_STA_0.M720 OR "DB356_M_UNIT_2_STA_0".M_CODES_UNIT_2_STA_0.M721,
                           M_FIXTURE_GRIPPER_OPEN := "DB356_M_UNIT_2_STA_0".M_CODES_UNIT_2_STA_0.M722 OR "DB356_M_UNIT_2_STA_0".M_CODES_UNIT_2_STA_0.M723,
                           UP_SEALING_STRUCTURE_CLOSED := "DB6800_UNIT_2_UP_SEALING_STRUCTURE".CLOSED,
                           DOWN_SEALING_STRUCTURE_CLOSED := "DB6801_UNIT_2_DOWN_SEALING_STRUCTURE".CLOSED,
                           PART_TYPE_FIXTURES := "DB7215_PART_TYPE".PART_TYPE_U02_FIXTURES,
                           ROBOT_PART_LOAD_UNLOAD := NOT "DB356_M_UNIT_2_STA_0".M_CODES_UNIT_2_STA_0.M50 AND NOT "DB356_M_UNIT_2_STA_0".M_CODES_UNIT_2_STA_0.M51,
                           ROBOT_OUT_OF_COLLISION := "DB7300_INTERLOCK_GENERAL".GENERAL_MACHINE.FROM_ROBOT_TO_UNIT_2.OUT_OF_COLLISION_MACHINE,
                           E_AXIS_HOME_POS := "DB5000_FIX_TABLE_POSITIONS".UNIT_2.AXIS_E20_HOME_POS,
                           W_AXIS_CLAMP_CHECK_POS := "DB154_CLADDING_AXIS_W21".SAFETY_POSITIONS.SAFETY_POSITION_4.IN_POSITION,
                           W_AXIS_UNCLAMP_CHECK_POS := "DB154_CLADDING_AXIS_W21".SAFETY_POSITIONS.SAFETY_POSITION_2.IN_POSITION,
                           UNIT_NO := 2,
                           FIXTURE_NO := 4,
                           NOT_CLAMPED_DURING_MACHINING_A => "DB426_ALARMS_WARNINGS".UNIT_02."720035",
                           PART_PRESENT_DISCORDANCY_A => "DB426_ALARMS_WARNINGS".UNIT_02."720011",
                           PART_TYPE_DISCORDANCY_A => "DB426_ALARMS_WARNINGS".UNIT_02."720003",
                           PART_TYPE_ORIENTATED_DISCORDANCY_A => "DB426_ALARMS_WARNINGS".UNIT_02."720027");
END_REGION

REGION Network 5: CALL FC3510 GRIPPERS
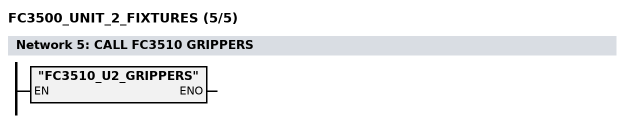
   RUNG wire#powerrail
      "FC3510_U2_GRIPPERS"()
   END_RUNG
   // the same network as SCL:
   "FC3510_U2_GRIPPERS"();
END_REGION
END_FUNCTION
